INTERFACE I_Parameter EXTENDS I_Disposable, I_Serializable, I_Deserializable, I_EventEmitter, I_HostMetadata

METHOD PUBLIC Accept
VAR_INPUT
	Visitor : I_ParameterVisitor;
END_VAR
END_METHOD

PROPERTY PUBLIC Data : I_DataType
GET
END_GET
END_PROPERTY

PROPERTY PUBLIC Name : T_MAXSTRING
GET
END_GET
END_PROPERTY

PROPERTY PUBLIC Parent : I_HostParameters
GET
END_GET
END_PROPERTY

END_INTERFACE

(* stored: Version 1.1.0.1, ProductVersion 3.1.4024.12
   Itf I_Parameter: Id {159f2e20-a209-4f39-91f2-c098c91b43ff}
   Method Accept: Id {b4082e10-8700-4a61-aff6-92b1cfe276e3}
   Property Data: Id {6cae52e4-0731-425f-97fa-fddac2574c0f}
   Get Get: Id {769812ad-118e-48c3-8d77-0b3e1561dc39}
   Property Name: Id {c8b1e40d-2c3c-4f6d-a049-feb5eac2bfd6}
   Get Get: Id {950a6e61-8a01-4fd1-bd13-b9ecae5fe260}
   Property Parent: Id {58629622-37e6-4b69-85c9-e36d0caa35e2}
   Get Get: Id {ad9817f8-b5e6-4e45-97ee-c8f74f650239} *)
